// Block: CTrk

DATA_BLOCK CTrk
VERSION : 0.1
   NON_RETAIN
   VAR
      Last_C_ID : DInt;
      Empty : CTrk_Item;
      A01_Preparation : CTrk_Item;
      A01_Processing : CTrk_Item;
      A02_Next : CTrk_Item;
      A02_Processing : CTrk_Item;
      A02_Consumed : CTrk_Item;
   END_VAR

BEGIN
   // No initialization required
END_DATA_BLOCK
